FUNCTION_BLOCK FB_ImmersionHeater EXTENDS FB_ComponentBase IMPLEMENTS I_HeatingElement
VAR
	_InSimulation : BOOL;
END_VAR

//{warning 'Add method implementation '}
METHOD CyclicLogic
IF _InSimulation THEN
	CyclicSimulate();
ELSE
	;
END_IF
END_METHOD

METHOD CyclicSimulate
VAR_INPUT
END_VAR
END_METHOD

PROPERTY InSimulation : BOOL
GET
InSimulation := _InSimulation;
END_GET
SET
_InSimulation := InSimulation;
END_SET
END_PROPERTY

{warning 'Add method implementation '}
METHOD Off : BOOL
END_METHOD

{warning 'Add method implementation '}
METHOD On : BOOL
END_METHOD

END_FUNCTION_BLOCK

(* stored: Version 1.1.0.1
   POU FB_ImmersionHeater: Id {919b0c87-9c83-4383-a90a-2f8eb0f0c477}, SpecialFunc None
   Method CyclicLogic: Id {45933a60-97dc-4460-9f93-d44e2be01b87}
   Method CyclicSimulate: Id {976eac1b-3866-4cc5-bd64-8eff3f359b98}
   Property InSimulation: Id {5acb5a22-956f-45a6-b0e6-4f08a4cb1ccd}
   Get Get: Id {4cfe8c45-336a-4db0-a934-ced2417e501d}
   Set Set: Id {d3682f48-cc9a-4205-985c-4b4fc0fb16e3}
   Method Off: Id {756579f5-dc61-48fe-a62c-510143c9686b}
   Method On: Id {167a6964-09ad-4d71-99ca-8e28f19c878e} *)
